FUNCTION_BLOCK JackRemoveWP (* Basic Function Block Type *)
  (* Standard: 61499-2 *)
  (* Version 0.0, 9/26/2018, dmidro, nxtControl GmbH, Template *)
  PACKAGE Main;
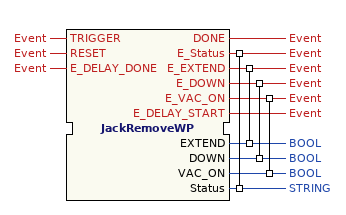
  EVENT_INPUT
    TRIGGER; (* Normal Execution Request *)
    RESET;
    E_DELAY_DONE;
  END_EVENT
  EVENT_OUTPUT
    DONE; (* Initialization Confirm *)
    E_Status WITH Status;
    E_EXTEND WITH EXTEND;
    E_DOWN WITH DOWN;
    E_VAC_ON WITH VAC_ON;
    E_DELAY_START;
  END_EVENT
  VAR_OUTPUT
    EXTEND : BOOL;
    DOWN : BOOL;
    VAC_ON : BOOL;
    Status : STRING;
  END_VAR
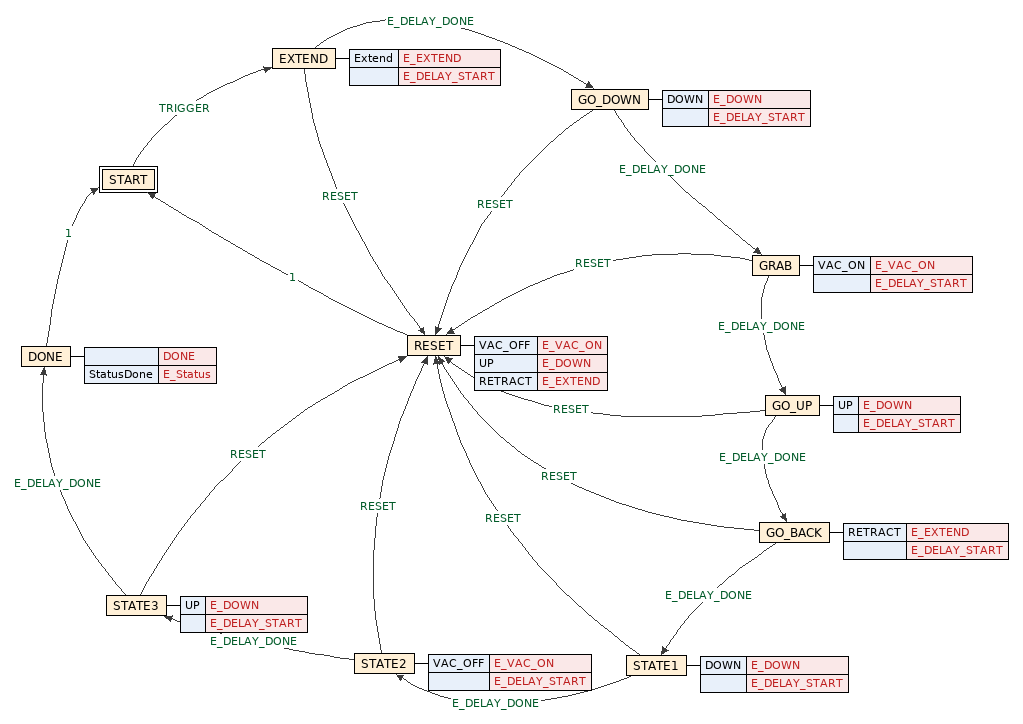
  EC_STATES
    START; (* Initial State *)
    GO_DOWN : DOWN -> E_DOWN, -> E_DELAY_START;
    GRAB : VAC_ON -> E_VAC_ON, -> E_DELAY_START;
    EXTEND : Extend -> E_EXTEND, -> E_DELAY_START;
    GO_BACK : RETRACT -> E_EXTEND, -> E_DELAY_START;
    GO_UP : UP -> E_DOWN, -> E_DELAY_START;
    DONE : -> DONE, StatusDone -> E_Status;
    RESET : VAC_OFF -> E_VAC_ON, UP -> E_DOWN, RETRACT -> E_EXTEND;
    STATE1 : DOWN -> E_DOWN, -> E_DELAY_START;
    STATE2 : VAC_OFF -> E_VAC_ON, -> E_DELAY_START;
    STATE3 : UP -> E_DOWN, -> E_DELAY_START;
  END_STATES
  EC_TRANSITIONS
    START TO EXTEND := TRIGGER;
    GO_DOWN TO GRAB := E_DELAY_DONE;
    GRAB TO GO_UP := E_DELAY_DONE;
    EXTEND TO GO_DOWN := E_DELAY_DONE;
    GO_BACK TO STATE1 := E_DELAY_DONE;
    GO_UP TO GO_BACK := E_DELAY_DONE;
    DONE TO START := 1;
    EXTEND TO RESET := RESET;
    GO_DOWN TO RESET := RESET;
    GRAB TO RESET := RESET;
    GO_UP TO RESET := RESET;
    GO_BACK TO RESET := RESET;
    RESET TO START := 1;
    STATE1 TO STATE2 := E_DELAY_DONE;
    STATE2 TO STATE3 := E_DELAY_DONE;
    STATE3 TO DONE := E_DELAY_DONE;
    STATE3 TO RESET := RESET;
    STATE2 TO RESET := RESET;
    STATE1 TO RESET := RESET;
  END_TRANSITIONS
  ALGORITHM INIT IN ST: (* Initialization algorithm *)
;
  END_ALGORITHM
  ALGORITHM REQ IN ST: (* Normally executed algorithm *)
;
  END_ALGORITHM
  ALGORITHM Extend IN ST:
EXTEND := TRUE;
E_DELAY_DONE := FALSE;
  END_ALGORITHM
  ALGORITHM DOWN IN ST:
DOWN := TRUE;
E_DELAY_DONE := FALSE;
  END_ALGORITHM
  ALGORITHM VAC_ON IN ST:
VAC_ON := TRUE;
E_DELAY_DONE := FALSE;
  END_ALGORITHM
  ALGORITHM UP IN ST:
DOWN := FALSE;
E_DELAY_DONE := FALSE;
  END_ALGORITHM
  ALGORITHM RETRACT IN ST:
EXTEND := FALSE;
E_DELAY_DONE := FALSE;
  END_ALGORITHM
  ALGORITHM VAC_OFF IN ST:
VAC_ON := FALSE;
E_DELAY_DONE := FALSE;
  END_ALGORITHM
  ALGORITHM StatusStarted IN ST:
Status := 'S';
  END_ALGORITHM
  ALGORITHM StatusDone IN ST:
Status := 'REMOVE_D';
E_DELAY_DONE := FALSE;
  END_ALGORITHM
END_FUNCTION_BLOCK
